FUNCTION_BLOCK CruiseControlObs
  (* Standard: 61499-2 *)
  (* Version 0.2, 2003-12-05, JHC, Rockwell Automation, Renamed from NEWCOMPFB. *)
  (* Version 0.1, 2002-01-08, JHC, Rockwell Automation, Added DLY FB as example. *)
  (* Version 0.0, 2000-05-27, JHC, Rockwell Automation *)
  (* Compiler header: package fb.rt.benchmarks.cruisecontrol; *)
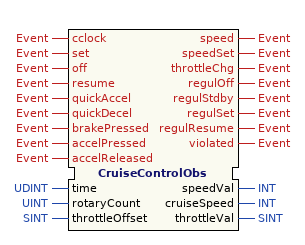
  EVENT_INPUT
    cclock;
    set;
    off;
    resume;
    quickAccel;
    quickDecel;
    brakePressed;
    accelPressed;
    accelReleased;
  END_EVENT
  EVENT_OUTPUT
    speed;
    speedSet;
    throttleChg;
    regulOff;
    regulStdby;
    regulSet;
    regulResume;
    violated;
  END_EVENT
  VAR_INPUT
    time : UDINT; (* 10ms tick *)
    rotaryCount : UINT;
    throttleOffset : SINT;
  END_VAR
  VAR_OUTPUT
    speedVal : INT; (* Output event qualifier *)
    cruiseSpeed : INT;
    throttleVal : SINT;
  END_VAR
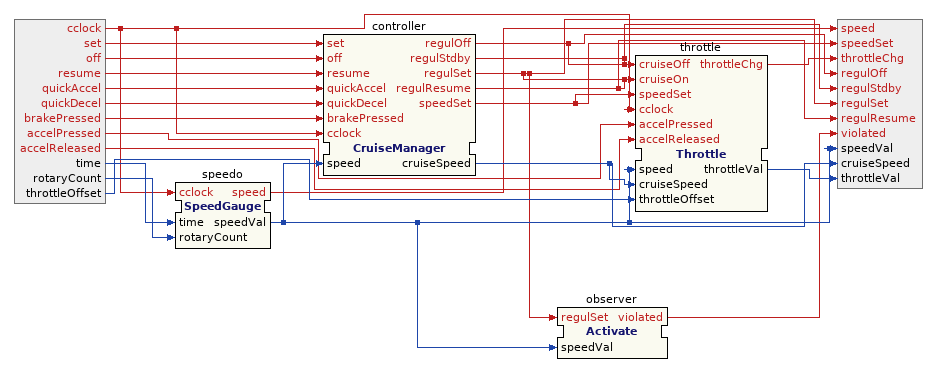
  FBS
    speedo : SpeedGauge;
    controller : CruiseManager;
    throttle : Throttle;
    observer : Activate;
  END_FBS
  EVENT_CONNECTIONS
    cclock TO speedo.cclock;
    speedo.speed TO speed;
    set TO controller.set;
    off TO controller.off;
    resume TO controller.resume;
    quickAccel TO controller.quickAccel;
    quickDecel TO controller.quickDecel;
    brakePressed TO controller.brakePressed;
    cclock TO controller.cclock;
    controller.regulOff TO throttle.cruiseOff;
    controller.regulStdby TO throttle.cruiseOff;
    controller.regulSet TO throttle.cruiseOn;
    controller.regulResume TO throttle.cruiseOn;
    controller.speedSet TO throttle.speedSet;
    controller.speedSet TO speedSet;
    cclock TO throttle.cclock;
    accelPressed TO throttle.accelPressed;
    accelReleased TO throttle.accelReleased;
    throttle.throttleChg TO throttleChg;
    controller.regulOff TO regulOff;
    controller.regulStdby TO regulStdby;
    controller.regulSet TO regulSet;
    controller.regulResume TO regulResume;
    controller.regulSet TO observer.regulSet;
    observer.violated TO violated;
  END_CONNECTIONS
  DATA_CONNECTIONS
    time TO speedo.time;
    rotaryCount TO speedo.rotaryCount;
    speedo.speedVal TO speedVal;
    speedo.speedVal TO controller.speed;
    speedo.speedVal TO throttle.speed;
    controller.cruiseSpeed TO throttle.cruiseSpeed;
    controller.cruiseSpeed TO cruiseSpeed;
    throttleOffset TO throttle.throttleOffset;
    throttle.throttleVal TO throttleVal;
    speedo.speedVal TO observer.speedVal;
  END_CONNECTIONS
END_FUNCTION_BLOCK
